// TIA Portal V19 export
DATA_BLOCK "DI_QF_WR02_03"   // DB31
// stored: AutoNumber false, InstanceOfName FB_QF, InstanceOfType FB
"FB_QF"
   // VAR RETAIN
   //    In { ExternalAccessible := 'False'; ExternalVisible := 'False'; ExternalWritable := 'False'} : Struct
   //       NotHalt : Bool;
   //       Auto : Bool;
   //       Hand : Bool;
   //       Tipp : Bool;
   //       T_WR02_zu_UE : Bool;
   //       T_WR02_zu_BE : Bool;
   //       T_WR03_zu_UE : Bool;
   //       T_WR03_zu_BE : Bool;
   //       S_WR02_lgsm_UE : Bool;
   //       S_WR02_lgsm_BE : Bool;
   //       S_WR03_lgsm_UE : Bool;
   //       S_WR03_lgsm_BE : Bool;
   //       S_WR02_UE : Bool;
   //       S_WR02_BE : Bool;
   //       S_WR03_UE : Bool;
   //       S_WR03_BE : Bool;
   //       Req_Ausfahrt_GO : Bool;
   //       Req_Aufgabe_GO : Bool;
   //       FU_betriebsbereit_WR02 : Bool;
   //       FU_betriebsbereit_WR03 : Bool;
   //       FU_Stoerung_WR02 : Bool;
   //       FU_Stoerung_WR03 : Bool;
   //       ErrQ : Bool;
   //       FU_speed_WR02 : Int;
   //       FU_speed_WR03 : Int;
   //    END_STRUCT;
   //    Param { ExternalAccessible := 'False'; ExternalVisible := 'False'; ExternalWritable := 'False'} : Struct
   //       "TO" : Time;
   //    END_STRUCT;
   //    Zst { ExternalAccessible := 'False'; ExternalVisible := 'False'; ExternalWritable := 'False'} : Struct
   //       Fehler : Bool;
   //       Req_WR02_In : Bool;
   //       Req_WR03_In : Bool;
   //       Req_WR02_Out : Bool;
   //       Req_WR03_Out : Bool;
   //       Tor_sicher : Bool;
   //       TW_sicher : Bool;
   //    END_STRUCT;
   //    Out { ExternalAccessible := 'False'; ExternalVisible := 'False'; ExternalWritable := 'False'} : Struct
   //       WR02_einfahren : Bool;
   //       WR02_ausfahren : Bool;
   //       WR03_einfahren : Bool;
   //       WR03_ausfahren : Bool;
   //       Soll_speed_WR02 : Int;
   //       Soll_speed_WR03 : Int;
   //    END_STRUCT;
   //    Mld { ExternalAccessible := 'False'; ExternalVisible := 'False'; ExternalWritable := 'False'} : Struct
   //       TO_WR02 : Bool;
   //       TO_WR03 : Bool;
   //       St_FU_WR02 : Bool;
   //       St_FU_WR03 : Bool;
   //       FU_nichtbereit_WR02 : Bool;
   //       FU_nichtbereit_WR03 : Bool;
   //       n_Auto : Bool;
   //       SF_WR02 : Bool;
   //       SF_WR03 : Bool;
   //    END_STRUCT;
   // END_VAR
   // VAR
   //    IEC_Timer { ExternalAccessible := 'False'; ExternalVisible := 'False'; ExternalWritable := 'False'} : Struct
   //       TO_WR02 { S7_SetPoint := 'True'} : TON_TIME;
   //       TO_WR03 { S7_SetPoint := 'True'} : TON_TIME;
   //    END_STRUCT;
   // END_VAR
BEGIN
END_DATA_BLOCK
